(* IEC 61131-3 sources: volt/packages/volt-lsp-iec/test-corpus/lenze-mid/Device/Plc Logic/Application/A71_LocalSources/ServoControl, 4 files *)

(* ---- BasicMotionControl.pou ---- *)
FUNCTION_BLOCK BasicMotionControl
VAR_INPUT
END_VAR
VAR_OUTPUT
END_VAR
VAR
END_VAR

%LANGUAGE LD
%NETWORK

END_FUNCTION_BLOCK

(* ---- FB_Lenze_i550.pou ---- *)
FUNCTION_BLOCK FB_Lenze_i550
VAR_INPUT
	iStatusWord : sUDT_FQIComm_Drive_Status;
	iGearRatioNumerator : REAL;
	iGearRatioDenominator : REAL;
	iNominalMotorSpeedwoSlipComp_RPM : REAL;
	iNominalMotorFrequency_Hz : REAL;
	iAxisJogSpeed_RPM : REAL;

END_VAR
VAR_OUTPUT
	oControlWord : sUDT_FQIComm_Drive_Control;
	oRefSpeed : WORD;

END_VAR
VAR
END_VAR
VAR_IN_OUT
	ioUDT			: UDT_FQI_Drive;
END_VAR
%LANGUAGE LD
%NETWORK
MOVE(EN := RAIL(), OPERAND('UINT_TO_WORD(ioUDT.Control.AutoSpeed)'), OUT => oRefSpeed);
%NETWORK
VAR w1 : ANY; END_VAR
w1 := TRUE;
ASSIGN(w1 AND iStatusWord.Bit3_Fault, Q => ioUDT.Status.Error);
ASSIGN(w1 AND INVERT(iStatusWord.Bit3_Fault) AND iStatusWord.Bit0_ReadyForOperation, Q => ioUDT.Status.DriveReady);
%NETWORK
VAR w2 : ANY; w3 : ANY; END_VAR
w2 := TRUE;
ASSIGN(w2 AND ioUDT.Control.Enable AND ioUDT.Control.StartAuto, Q => oControlWord.Bit4_RunForward);
w3 := w2 AND ioUDT.Control.ResetError;
ASSIGN(w3, Q => oControlWord.Bit7_ResetFault);
ASSIGN(w3, Q_RESET => ioUDT.Control.ResetError);
ASSIGN(w2 AND ioUDT.Control.Reverse, Q => oControlWord.Bit12_ReverseDirection);

END_FUNCTION_BLOCK

(* ---- ServoControl.pou ---- *)
FUNCTION_BLOCK ServoControl
VAR_INPUT
	iServoStatus 	: sUDT_ServoComm_Drive_Status;
	iEnableHomeMovement : BOOL;
	iEnablePower 		: BOOL;
	iFF100ms 			: BOOL;

END_VAR
VAR_OUTPUT
	oServoControl 		: sUDT_ServoComm_Drive_Control;

END_VAR
VAR

	intYScale: 	INT;

	Man_SetHomePos: BOOL;
	OSP_SetHomnePos: R_TRIG;
	HomingDoneDelay: TON;
END_VAR
VAR_IN_OUT
	ioUDT_ServoDrive			: UDT_ServoDrive;
END_VAR
VAR RETAIN PERSISTENT
	STATE_Prehoming: BOOL;
	STATE_HomePosNOK: BOOL;
	STATE_HomePOSOK: BOOL;
	STATE_WaitingForEnable: BOOL;
	STATE_Synchronising: BOOL;
END_VAR
VAR CONSTANT
	ctCurveIs0ToMax: INT := 0;
	ctCurveIs0To0: INT := 1;
	ctCurveIsSpeed: INT := 2;
END_VAR
%LANGUAGE LD
%NETWORK "Network 2 : Initialise with STATE HomePosNotOK"
VAR w1 : ANY; END_VAR
w1 := INVERT(STATE_Prehoming) AND INVERT(STATE_HomePosNOK) AND INVERT(STATE_HomePOSOK) AND INVERT(STATE_WaitingForEnable) AND INVERT(STATE_Synchronising);
ASSIGN(w1, Q_RESET => STATE_Prehoming);
ASSIGN(w1, Q_RESET => STATE_HomePosNOK);
ASSIGN(w1, Q_RESET => STATE_HomePOSOK);
ASSIGN(w1, Q_RESET => STATE_WaitingForEnable);
ASSIGN(w1, Q_RESET => STATE_Synchronising);
ASSIGN(w1, Q_SET => STATE_HomePosNOK);
%NETWORK "Network 3 : STATE: Prehoming "
ASSIGN((STATE_WaitingForEnable OR STATE_Synchronising) AND iServoStatus.DriveCommAlive AND Man_SetHomePos AND iServoStatus.HomingPosOK, Q_SET => STATE_Prehoming, Q_RESET => STATE_HomePOSOK, Q_RESET => STATE_WaitingForEnable, Q_RESET => STATE_Synchronising);
%NETWORK "STATE: HomePos not OK"
ASSIGN((STATE_Prehoming OR STATE_HomePOSOK OR STATE_WaitingForEnable OR STATE_Synchronising) AND iServoStatus.DriveCommAlive AND INVERT(iServoStatus.HomingPosOK), Q_SET => STATE_HomePosNOK, Q_RESET => STATE_Prehoming, Q_RESET => STATE_HomePOSOK, Q_RESET => STATE_WaitingForEnable, Q_RESET => STATE_Synchronising);
%NETWORK "Network 5: STATE: HomePos OK"
ASSIGN(STATE_HomePosNOK AND iServoStatus.DriveCommAlive AND iServoStatus.HomingPosOK, Q_SET => STATE_HomePOSOK, Q_RESET => STATE_HomePosNOK, Q_RESET => Man_SetHomePos);
%NETWORK "Network 6 : STATE: WaitingForEnable"
ASSIGN(STATE_HomePOSOK OR STATE_Synchronising AND INVERT(ioUDT_ServoDrive.Control.SetDriveEnable), Q_SET => STATE_WaitingForEnable, Q_RESET => STATE_HomePOSOK, Q_RESET => STATE_Synchronising);
%NETWORK "DONE Network 7: STATE: Synchronising"
ASSIGN(STATE_WaitingForEnable AND ioUDT_ServoDrive.Control.SetDriveEnable, Q_SET => STATE_Synchronising, Q_RESET => STATE_WaitingForEnable);
%NETWORK "DONE Network 8: Activate set HomePos Cycle"
VAR w2 : ANY; END_VAR
w2 := OSP_SetHomnePos(CLK := ioUDT_ServoDrive.Control.StartSetHomePos AND ioUDT_ServoDrive.Status.DriveIsReady);
ASSIGN(w2, Q_SET => Man_SetHomePos);
ASSIGN(w2, Q_RESET => ioUDT_ServoDrive.Control.StartSetHomePos);
%NETWORK "DONE Network 9: Output: Activate Synchronise drive"
ASSIGN(STATE_Synchronising AND ioUDT_ServoDrive.Control.SetInSync, Q => oServoControl.ActivateCamming);
%NETWORK "DONE Network 10: Reset HomePos in Servo drive"
ASSIGN(STATE_Prehoming AND Man_SetHomePos, Q => oServoControl.ResetHomePos);
%NETWORK "DONE Network 11: Set HomePos in Servo drive"
ASSIGN(STATE_HomePosNOK AND Man_SetHomePos AND iEnableHomeMovement AND ioUDT_ServoDrive.Status.DriveIsReady, Q => oServoControl.SetHomePos);
%NETWORK "DONE Network 11: Set HomePos in Servo drive"
ASSIGN(ioUDT_ServoDrive.Control.SetBrakeRelease, Q => oServoControl.ReleaseBrake);
%NETWORK "TODO Network 16: Enable drive from software"
ASSIGN(ioUDT_ServoDrive.Control.SetDriveEnable AND iEnablePower, Q => oServoControl.Enable);
%NETWORK "DONE Network 17: Reset error"
ASSIGN(ioUDT_ServoDrive.Control.ResetError AND iFF100ms, Q => oServoControl.ResetError);
%NETWORK "DONE Network 18: SelectBypassCAM"
ASSIGN(ioUDT_ServoDrive.Control.SelectBypassCAM, Q => oServoControl.SelectBypassCAM);
%NETWORK "DONE Network 19: Output: X-offset"
EXECUTE(EN := RAIL(), 'ioUDT_ServoDrive.CAM.X_Offset_ToSlave := ioUDT_ServoDrive.CAM.X_Offset_FromMaster + ioUDT_ServoDrive.CAM.X_Offset_Recipe;
oServoControl.XOffset := INT_TO_WORD(ioUDT_ServoDrive.CAM.X_Offset_Base + ioUDT_ServoDrive.CAM.X_Offset_ToSlave);');
%NETWORK "DONE Network 20: Scaling of the Y value"
VAR w3 : ANY; END_VAR
w3 := True;
MOVE(EN := GE(EN := w3, ioUDT_ServoDrive.CAM.CamType, ctCurveIs0ToMax).OUT, 1000, OUT => oServoControl.YScale);
ADD(EN := OR(GE(EN := w3, ioUDT_ServoDrive.CAM.CamType, ctCurveIs0To0).OUT, GE(EN := RAIL(), ioUDT_ServoDrive.CAM.CamType, ctCurveIsSpeed).OUT), ioUDT_ServoDrive.CAM.Y_Scale_Base, ioUDT_ServoDrive.CAM.Y_Scale_Recipe, OUT => oServoControl.YScale);
%NETWORK "DONE Network 21: Y-offset"
EXECUTE(EN := RAIL(), 'oServoControl.YOffset := INT_TO_WORD(ioUDT_ServoDrive.CAM.Y_Offset_Base + ioUDT_ServoDrive.CAM.Y_Offset_Recipe);');
%NETWORK "TODO Network 22: Status inputs from drive"
%NETWORK "TODO Network 23: SetOuput bits to drive"
%NETWORK "DONE Network 24: Output to Program"
VAR w4 : ANY; END_VAR
w4 := True;
ASSIGN(w4 AND iServoStatus.ReadyForMotion, Q => ioUDT_ServoDrive.Status.DriveIsReady);
ASSIGN(w4 AND iServoStatus.InSync, Q => ioUDT_ServoDrive.Status.InSync);
ASSIGN(w4 AND iServoStatus.TorqueLimit, Q => ioUDT_ServoDrive.Status.DriveTorqueError);
ASSIGN(HomingDoneDelay(IN := w4 AND INVERT(STATE_Prehoming) AND INVERT(STATE_HomePosNOK), PT := T#2S), Q => ioUDT_ServoDrive.Status.DriveIsHomed);
%NETWORK "DONE Network 25: ActualXPos/Ypos"
MOVE(EN := RAIL(), OPERAND('LREAL_TO_INT(iServoStatus.ActPos)'), OUT => ioUDT_ServoDrive.CAM.ActualYPos);
%NETWORK "DONE Network 26: ActualSpeed"
MOVE(EN := RAIL(), OPERAND('LREAL_TO_INT(iServoStatus.ActSpeed)'), OUT => ioUDT_ServoDrive.CAM.ActualYSpeed);
%NETWORK
MOVE(EN := RAIL(), ioUDT_ServoDrive.Control.TorqueLimit, OUT => oServoControl.TorqueLimit);
%NETWORK "DONE Network 27: Reset ResetError in UDT"
ASSIGN(True AND ioUDT_ServoDrive.Status.DriveIsReady, Q_RESET => ioUDT_ServoDrive.Control.ResetError);

END_FUNCTION_BLOCK

(* ---- VirtualMasterControl.pou ---- *)
FUNCTION_BLOCK VirtualMasterControl
VAR_INPUT
	iAcc: REAL:=1800;
	iDec: REAL:=1800;

END_VAR
VAR_OUTPUT
END_VAR
VAR
END_VAR
VAR_IN_OUT
	ioVirtualMaster: UDT_VirtualMaster;
	ioVirtualMasterCom: sUDT_VirtualMasterComm_Drive;

END_VAR

%LANGUAGE LD
%NETWORK
VAR w1 : ANY; END_VAR
w1 := TRUE;
ASSIGN(w1 AND ioVirtualMaster.Control.SetDriveEnable, Q => ioVirtualMasterCom.Control.Enable);
ASSIGN(w1 AND ioVirtualMaster.Control.ResetError, Q => ioVirtualMasterCom.Control.ResetError);
%NETWORK
VAR w2 : ANY; END_VAR
w2 := ioVirtualMaster.Control.StartMovement;
ASSIGN(w2, Q => ioVirtualMasterCom.Control.StartMovement);
MOVE(EN := w2, Mach1_Data.Drives.MainDrive_VM.Control.DriveMasterSpeed, OUT => ioVirtualMasterCom.Control.VelUnit);
MOVE(EN := w2, iDec, OUT => ioVirtualMasterCom.Control.DecUnit);
MOVE(EN := w2, iAcc, OUT => ioVirtualMasterCom.Control.AccUnit);
%NETWORK
DIV(EN := DIV(EN := TRUE, OPERAND('LREAL_TO_INT(ioVirtualMasterCom.Status.ActSpeed)'), 6, OUT => ioVirtualMaster.Status.ActSpeed), OPERAND('LREAL_TO_INT(ioVirtualMasterCom.Status.ActPos)'), 1, OUT => ioVirtualMaster.Status.ActXPos);
%NETWORK
ASSIGN(ioVirtualMasterCom.Status.ReadyForMotion, Q => ioVirtualMaster.Status.DriveIsReady);
%NETWORK

END_FUNCTION_BLOCK
